// TIA Portal project "TestCase3_S1500_Met_Fouten" (V18)

(* hardware
DEVICE "S7-1500/ET200MP station_1"  S7-1500 station
   slot 0: "Rail_0"  Rack  6ES7 590-1***0-0AA0
   slot 1: "PLC_1"  CPU 1511C-1 PN  6ES7 511-1CK00-0AB0  V2.9
      slot 3: "CPU display_1"  6ES7591-1AA00-0AA0
      slot 32768: "PROFINET interface_1"  X1
         slot 32769: "Port_1"  X1 P1
         slot 32770: "Port_2"  X1 P2
      slot 34817: "Virtual CP interface port_1"  Virtual CP interface port  Virtual CP interface port
*)

// ===== PLC "PLC_1"  CPU 1511C-1 PN =====

DATA_BLOCK "Data_block_1"   // DB1
{ S7_Optimized_Access := 'FALSE' }
VERSION : 0.1
   VAR
      "A" : Bool;
      "B" : Int;
      C : Int;
   END_VAR
BEGIN
END_DATA_BLOCK

DATA_BLOCK "Data_block_2"   // DB2
{ S7_Optimized_Access := 'FALSE' }
VERSION : 0.1
   VAR
      "A" : Byte;
      "B" : Word;
      C : DWord;
      D : Int;
      "E" : DInt;
      F : Real;
   END_VAR
BEGIN
END_DATA_BLOCK

ORGANIZATION_BLOCK "Main"   // OB1, FBD, ProgramCycle
TITLE = "Main Program Sweep (Cycle)"
{ S7_Optimized_Access := 'FALSE' }
VERSION : 0.1
   VAR_TEMP
      EV_CLASS : Byte;   // Bits 0-3 = 1:Coming event, Bits 4-7 = 1:Event class 1
      SCAN_1 : Byte;   // 1:Initial call of the OB, 3: Call 2-n of the OB
      PRIORITY : Byte;   // Priority of OB Execution
      OB_NUMBR : Byte;   // OB number
      RESERVED_1 : Byte;   // Reserved for system
      RESERVED_2 : Byte;   // Reserved for system
      PREV_CYCLE : Int;   // Previous program cycle time (milliseconds)
      MIN_CYCLE : Int;   // Minimum program cycle time (milliseconds)
      MAX_CYCLE : Int;   // Maximum program cycle time (milliseconds)
      DATE_TIME : Date_And_Time;   // Date and time OB started
   END_VAR
   VAR_TEMP   // added for the SCL form of the ladder/FBD networks
      _w1 : Bool;
   END_VAR
BEGIN

REGION Network 1
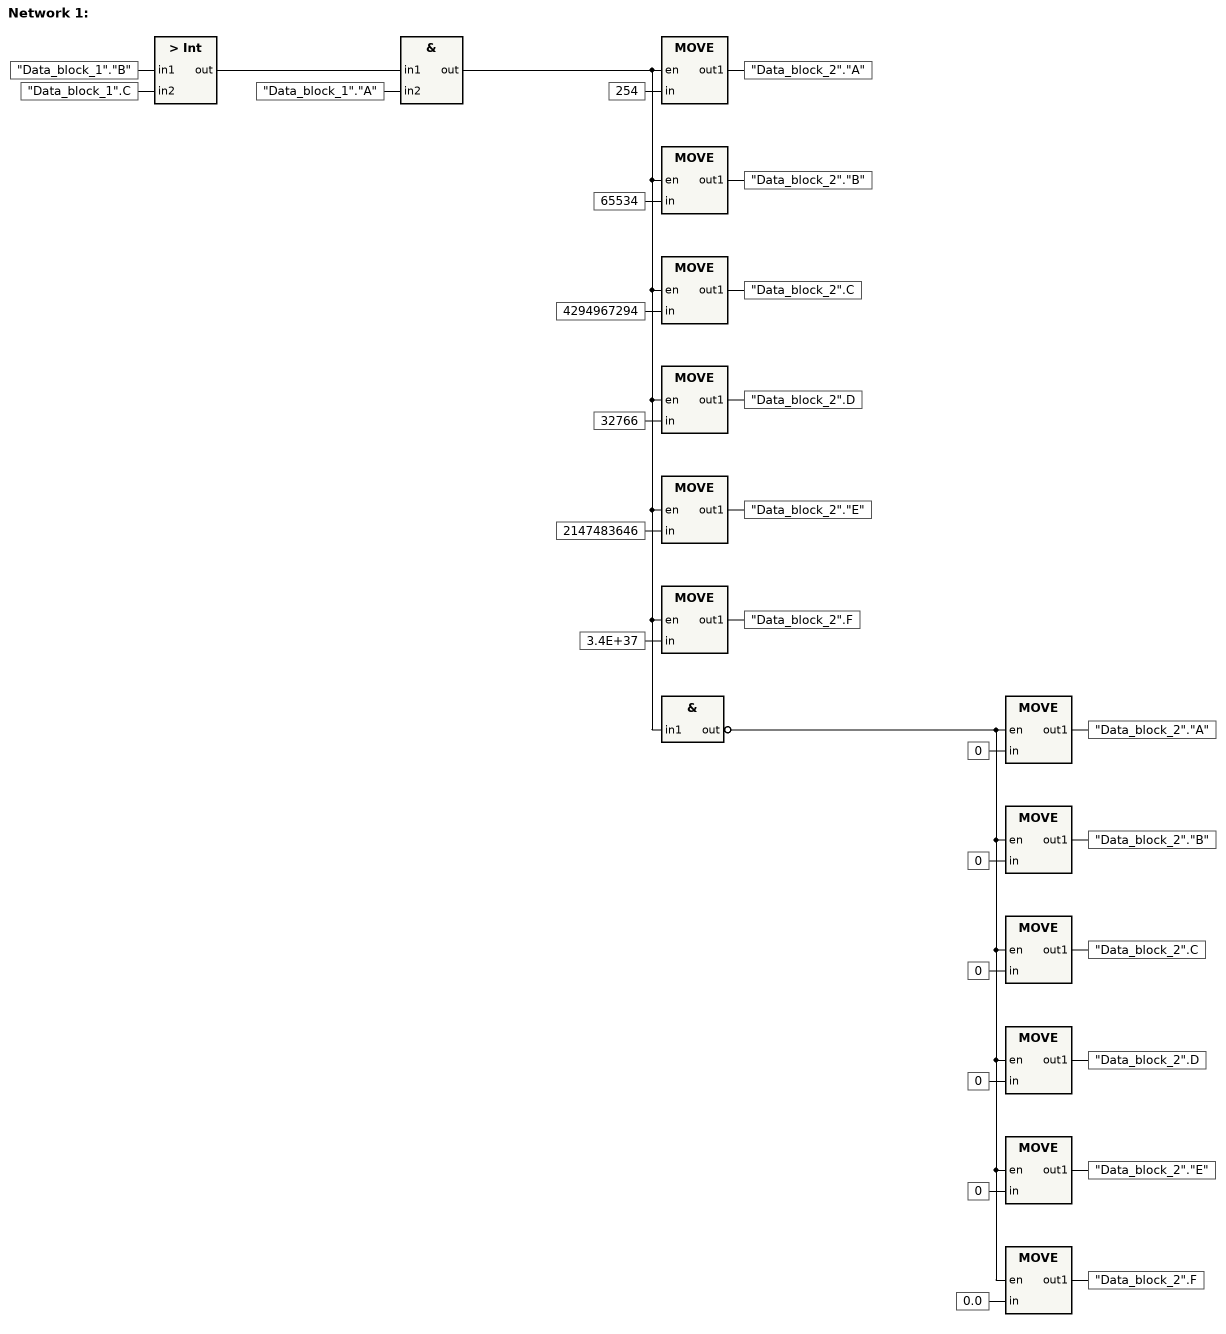
   #_w1 := ("Data_block_1"."B" > "Data_block_1".C) AND "Data_block_1"."A";
   IF #_w1 THEN
       "Data_block_2"."A" := 254;
       "Data_block_2"."B" := 65534;
       "Data_block_2".C := 4294967294;
       "Data_block_2".D := 32766;
       "Data_block_2"."E" := 2147483646;
       "Data_block_2".F := 3.4E+37;
   END_IF;
   IF NOT #_w1 THEN
       "Data_block_2"."A" := 0;
       "Data_block_2"."B" := 0;
       "Data_block_2".C := 0;
       "Data_block_2".D := 0;
       "Data_block_2"."E" := 0;
       "Data_block_2".F := 0.0;
   END_IF;
END_REGION
END_ORGANIZATION_BLOCK